(* IEC 61131-3 sources: AXOpen/src/components.keyence.vision/ctrl/src/Axo_IV3 (part 3) *)

            //*************************ToolResult_33*************************
            _retVal := Siemens.Simatic.DistributedIO.ReadData((Config.HWIDs.HwID_ToolResult_33) ,_data_in);
            IF _retVal > WORD#0 THEN
                Messenger.Activate(UINT#1638, eAxoMessageCategory#Error);
                Status.Error.Id := UINT#1638;
                RETURN;
            END_IF;

            _word.%B0 := _data_in[1];
            _word.%B1 := _data_in[0];
            Inputs.ToolResult_33.MatchingRate       :=  TO_UINT(_word);        // IW712
            _word.%B0 := _data_in[3];
            _word.%B1 := _data_in[2];
            Inputs.ToolResult_33.MatchingRateMAX    :=  TO_UINT(_word);        // IW714
            _word.%B0 := _data_in[5];
            _word.%B1 := _data_in[4];
            Inputs.ToolResult_33.MatchingRateMIN    :=  TO_UINT(_word);        // IW716
            _word.%B0 := _data_in[7];
            _word.%B1 := _data_in[6];
            Inputs.ToolResult_33.LowerThreshold     :=  TO_UINT(_word);        // IW718
            _word.%B0 := _data_in[9];
            _word.%B1 := _data_in[8];
            Inputs.ToolResult_33.UpperThreshold     :=  TO_UINT(_word);        // IW720
            _word.%B0 := _data_in[11];
            _word.%B1 := _data_in[10];
            Inputs.ToolResult_33.DecimalPointPosition:=  TO_UINT(_word);       // IW722
            _word.%B0 := _data_in[13];
            _word.%B1 := _data_in[12];
            Inputs.ToolResult_33.Data_1             :=  TO_UINT(_word);        // IW724
            _word.%B0 := _data_in[15];
            _word.%B1 := _data_in[14];
            Inputs.ToolResult_33.Data_2             :=  TO_UINT(_word);        // IW726
            _word.%B0 := _data_in[17];
            _word.%B1 := _data_in[16];
            Inputs.ToolResult_33.Data_3             :=  TO_UINT(_word);        // IW728
                                                                                    // IW730
            //***************************************************************

            //*************************ToolResult_34*************************
            _retVal := Siemens.Simatic.DistributedIO.ReadData((Config.HWIDs.HwID_ToolResult_34) ,_data_in);
            IF _retVal > WORD#0 THEN
                Messenger.Activate(UINT#1639, eAxoMessageCategory#Error);
                Status.Error.Id := UINT#1639;
                RETURN;
            END_IF;

            _word.%B0 := _data_in[1];
            _word.%B1 := _data_in[0];
            Inputs.ToolResult_34.MatchingRate       :=  TO_UINT(_word);        // IW732
            _word.%B0 := _data_in[3];
            _word.%B1 := _data_in[2];
            Inputs.ToolResult_34.MatchingRateMAX    :=  TO_UINT(_word);        // IW734
            _word.%B0 := _data_in[5];
            _word.%B1 := _data_in[4];
            Inputs.ToolResult_34.MatchingRateMIN    :=  TO_UINT(_word);        // IW736
            _word.%B0 := _data_in[7];
            _word.%B1 := _data_in[6];
            Inputs.ToolResult_34.LowerThreshold     :=  TO_UINT(_word);        // IW738
            _word.%B0 := _data_in[9];
            _word.%B1 := _data_in[8];
            Inputs.ToolResult_34.UpperThreshold     :=  TO_UINT(_word);        // IW740
            _word.%B0 := _data_in[11];
            _word.%B1 := _data_in[10];
            Inputs.ToolResult_34.DecimalPointPosition:=  TO_UINT(_word);       // IW742
            _word.%B0 := _data_in[13];
            _word.%B1 := _data_in[12];
            Inputs.ToolResult_34.Data_1             :=  TO_UINT(_word);        // IW744
            _word.%B0 := _data_in[15];
            _word.%B1 := _data_in[14];
            Inputs.ToolResult_34.Data_2             :=  TO_UINT(_word);        // IW746
            _word.%B0 := _data_in[17];
            _word.%B1 := _data_in[16];
            Inputs.ToolResult_34.Data_3             :=  TO_UINT(_word);        // IW748
                                                                                    // IW750
            //***************************************************************

            //*************************ToolResult_35*************************
            _retVal := Siemens.Simatic.DistributedIO.ReadData((Config.HWIDs.HwID_ToolResult_35) ,_data_in);
            IF _retVal > WORD#0 THEN
                Messenger.Activate(UINT#1640, eAxoMessageCategory#Error);
                Status.Error.Id := UINT#1640;
                RETURN;
            END_IF;

            _word.%B0 := _data_in[1];
            _word.%B1 := _data_in[0];
            Inputs.ToolResult_35.MatchingRate       :=  TO_UINT(_word);        // IW752
            _word.%B0 := _data_in[3];
            _word.%B1 := _data_in[2];
            Inputs.ToolResult_35.MatchingRateMAX    :=  TO_UINT(_word);        // IW754
            _word.%B0 := _data_in[5];
            _word.%B1 := _data_in[4];
            Inputs.ToolResult_35.MatchingRateMIN    :=  TO_UINT(_word);        // IW756
            _word.%B0 := _data_in[7];
            _word.%B1 := _data_in[6];
            Inputs.ToolResult_35.LowerThreshold     :=  TO_UINT(_word);        // IW758
            _word.%B0 := _data_in[9];
            _word.%B1 := _data_in[8];
            Inputs.ToolResult_35.UpperThreshold     :=  TO_UINT(_word);        // IW760
            _word.%B0 := _data_in[11];
            _word.%B1 := _data_in[10];
            Inputs.ToolResult_35.DecimalPointPosition:=  TO_UINT(_word);       // IW762
            _word.%B0 := _data_in[13];
            _word.%B1 := _data_in[12];
            Inputs.ToolResult_35.Data_1             :=  TO_UINT(_word);        // IW764
            _word.%B0 := _data_in[15];
            _word.%B1 := _data_in[14];
            Inputs.ToolResult_35.Data_2             :=  TO_UINT(_word);        // IW766
            _word.%B0 := _data_in[17];
            _word.%B1 := _data_in[16];
            Inputs.ToolResult_35.Data_3             :=  TO_UINT(_word);        // IW768
                                                                                    // IW770
            //***************************************************************

            //*************************ToolResult_36*************************
            _retVal := Siemens.Simatic.DistributedIO.ReadData((Config.HWIDs.HwID_ToolResult_36) ,_data_in);
            IF _retVal > WORD#0 THEN
                Messenger.Activate(UINT#1641, eAxoMessageCategory#Error);
                Status.Error.Id := UINT#1641;
                RETURN;
            END_IF;

            _word.%B0 := _data_in[1];
            _word.%B1 := _data_in[0];
            Inputs.ToolResult_36.MatchingRate       :=  TO_UINT(_word);        // IW772
            _word.%B0 := _data_in[3];
            _word.%B1 := _data_in[2];
            Inputs.ToolResult_36.MatchingRateMAX    :=  TO_UINT(_word);        // IW774
            _word.%B0 := _data_in[5];
            _word.%B1 := _data_in[4];
            Inputs.ToolResult_36.MatchingRateMIN    :=  TO_UINT(_word);        // IW776
            _word.%B0 := _data_in[7];
            _word.%B1 := _data_in[6];
            Inputs.ToolResult_36.LowerThreshold     :=  TO_UINT(_word);        // IW778
            _word.%B0 := _data_in[9];
            _word.%B1 := _data_in[8];
            Inputs.ToolResult_36.UpperThreshold     :=  TO_UINT(_word);        // IW780
            _word.%B0 := _data_in[11];
            _word.%B1 := _data_in[10];
            Inputs.ToolResult_36.DecimalPointPosition:=  TO_UINT(_word);       // IW782
            _word.%B0 := _data_in[13];
            _word.%B1 := _data_in[12];
            Inputs.ToolResult_36.Data_1             :=  TO_UINT(_word);        // IW784
            _word.%B0 := _data_in[15];
            _word.%B1 := _data_in[14];
            Inputs.ToolResult_36.Data_2             :=  TO_UINT(_word);        // IW786
            _word.%B0 := _data_in[17];
            _word.%B1 := _data_in[16];
            Inputs.ToolResult_36.Data_3             :=  TO_UINT(_word);        // IW788
                                                                                    // IW790
            //***************************************************************

            //*************************ToolResult_37*************************
            _retVal := Siemens.Simatic.DistributedIO.ReadData((Config.HWIDs.HwID_ToolResult_37) ,_data_in);
            IF _retVal > WORD#0 THEN
                Messenger.Activate(UINT#1642, eAxoMessageCategory#Error);
                Status.Error.Id := UINT#1642;
                RETURN;
            END_IF;

            _word.%B0 := _data_in[1];
            _word.%B1 := _data_in[0];
            Inputs.ToolResult_37.MatchingRate       :=  TO_UINT(_word);        // IW792
            _word.%B0 := _data_in[3];
            _word.%B1 := _data_in[2];
            Inputs.ToolResult_37.MatchingRateMAX    :=  TO_UINT(_word);        // IW794
            _word.%B0 := _data_in[5];
            _word.%B1 := _data_in[4];
            Inputs.ToolResult_37.MatchingRateMIN    :=  TO_UINT(_word);        // IW796
            _word.%B0 := _data_in[7];
            _word.%B1 := _data_in[6];
            Inputs.ToolResult_37.LowerThreshold     :=  TO_UINT(_word);        // IW798
            _word.%B0 := _data_in[9];
            _word.%B1 := _data_in[8];
            Inputs.ToolResult_37.UpperThreshold     :=  TO_UINT(_word);        // IW800
            _word.%B0 := _data_in[11];
            _word.%B1 := _data_in[10];
            Inputs.ToolResult_37.DecimalPointPosition:=  TO_UINT(_word);       // IW802
            _word.%B0 := _data_in[13];
            _word.%B1 := _data_in[12];
            Inputs.ToolResult_37.Data_1             :=  TO_UINT(_word);        // IW804
            _word.%B0 := _data_in[15];
            _word.%B1 := _data_in[14];
            Inputs.ToolResult_37.Data_2             :=  TO_UINT(_word);        // IW806
            _word.%B0 := _data_in[17];
            _word.%B1 := _data_in[16];
            Inputs.ToolResult_37.Data_3             :=  TO_UINT(_word);        // IW808
                                                                                    // IW810
            //***************************************************************

            //*************************ToolResult_38*************************
            _retVal := Siemens.Simatic.DistributedIO.ReadData((Config.HWIDs.HwID_ToolResult_38) ,_data_in);
            IF _retVal > WORD#0 THEN
                Messenger.Activate(UINT#1643, eAxoMessageCategory#Error);
                Status.Error.Id := UINT#1643;
                RETURN;
            END_IF;

            _word.%B0 := _data_in[1];
            _word.%B1 := _data_in[0];
            Inputs.ToolResult_38.MatchingRate       :=  TO_UINT(_word);        // IW812
            _word.%B0 := _data_in[3];
            _word.%B1 := _data_in[2];
            Inputs.ToolResult_38.MatchingRateMAX    :=  TO_UINT(_word);        // IW814
            _word.%B0 := _data_in[5];
            _word.%B1 := _data_in[4];
            Inputs.ToolResult_38.MatchingRateMIN    :=  TO_UINT(_word);        // IW816
            _word.%B0 := _data_in[7];
            _word.%B1 := _data_in[6];
            Inputs.ToolResult_38.LowerThreshold     :=  TO_UINT(_word);        // IW818
            _word.%B0 := _data_in[9];
            _word.%B1 := _data_in[8];
            Inputs.ToolResult_38.UpperThreshold     :=  TO_UINT(_word);        // IW820
            _word.%B0 := _data_in[11];
            _word.%B1 := _data_in[10];
            Inputs.ToolResult_38.DecimalPointPosition:=  TO_UINT(_word);       // IW822
            _word.%B0 := _data_in[13];
            _word.%B1 := _data_in[12];
            Inputs.ToolResult_38.Data_1             :=  TO_UINT(_word);        // IW824
            _word.%B0 := _data_in[15];
            _word.%B1 := _data_in[14];
            Inputs.ToolResult_38.Data_2             :=  TO_UINT(_word);        // IW826
            _word.%B0 := _data_in[17];
            _word.%B1 := _data_in[16];
            Inputs.ToolResult_38.Data_3             :=  TO_UINT(_word);        // IW828
                                                                                    // IW830
            //***************************************************************

            //*************************ToolResult_39*************************
            _retVal := Siemens.Simatic.DistributedIO.ReadData((Config.HWIDs.HwID_ToolResult_39) ,_data_in);
            IF _retVal > WORD#0 THEN
                Messenger.Activate(UINT#1644, eAxoMessageCategory#Error);
                Status.Error.Id := UINT#1644;
                RETURN;
            END_IF;

            _word.%B0 := _data_in[1];
            _word.%B1 := _data_in[0];
            Inputs.ToolResult_39.MatchingRate       :=  TO_UINT(_word);        // IW832
            _word.%B0 := _data_in[3];
            _word.%B1 := _data_in[2];
            Inputs.ToolResult_39.MatchingRateMAX    :=  TO_UINT(_word);        // IW834
            _word.%B0 := _data_in[5];
            _word.%B1 := _data_in[4];
            Inputs.ToolResult_39.MatchingRateMIN    :=  TO_UINT(_word);        // IW836
            _word.%B0 := _data_in[7];
            _word.%B1 := _data_in[6];
            Inputs.ToolResult_39.LowerThreshold     :=  TO_UINT(_word);        // IW838
            _word.%B0 := _data_in[9];
            _word.%B1 := _data_in[8];
            Inputs.ToolResult_39.UpperThreshold     :=  TO_UINT(_word);        // IW840
            _word.%B0 := _data_in[11];
            _word.%B1 := _data_in[10];
            Inputs.ToolResult_39.DecimalPointPosition:=  TO_UINT(_word);       // IW842
            _word.%B0 := _data_in[13];
            _word.%B1 := _data_in[12];
            Inputs.ToolResult_39.Data_1             :=  TO_UINT(_word);        // IW844
            _word.%B0 := _data_in[15];
            _word.%B1 := _data_in[14];
            Inputs.ToolResult_39.Data_2             :=  TO_UINT(_word);        // IW846
            _word.%B0 := _data_in[17];
            _word.%B1 := _data_in[16];
            Inputs.ToolResult_39.Data_3             :=  TO_UINT(_word);        // IW848
                                                                                    // IW850
            //***************************************************************

            //*************************ToolResult_40*************************
            _retVal := Siemens.Simatic.DistributedIO.ReadData((Config.HWIDs.HwID_ToolResult_40) ,_data_in);
            IF _retVal > WORD#0 THEN
                Messenger.Activate(UINT#1645, eAxoMessageCategory#Error);
                Status.Error.Id := UINT#1645;
                RETURN;
            END_IF;

            _word.%B0 := _data_in[1];
            _word.%B1 := _data_in[0];
            Inputs.ToolResult_40.MatchingRate       :=  TO_UINT(_word);        // IW852
            _word.%B0 := _data_in[3];
            _word.%B1 := _data_in[2];
            Inputs.ToolResult_40.MatchingRateMAX    :=  TO_UINT(_word);        // IW854
            _word.%B0 := _data_in[5];
            _word.%B1 := _data_in[4];
            Inputs.ToolResult_40.MatchingRateMIN    :=  TO_UINT(_word);        // IW856
            _word.%B0 := _data_in[7];
            _word.%B1 := _data_in[6];
            Inputs.ToolResult_40.LowerThreshold     :=  TO_UINT(_word);        // IW858
            _word.%B0 := _data_in[9];
            _word.%B1 := _data_in[8];
            Inputs.ToolResult_40.UpperThreshold     :=  TO_UINT(_word);        // IW860
            _word.%B0 := _data_in[11];
            _word.%B1 := _data_in[10];
            Inputs.ToolResult_40.DecimalPointPosition:=  TO_UINT(_word);       // IW862
            _word.%B0 := _data_in[13];
            _word.%B1 := _data_in[12];
            Inputs.ToolResult_40.Data_1             :=  TO_UINT(_word);        // IW864
            _word.%B0 := _data_in[15];
            _word.%B1 := _data_in[14];
            Inputs.ToolResult_40.Data_2             :=  TO_UINT(_word);        // IW866
            _word.%B0 := _data_in[17];
            _word.%B1 := _data_in[16];
            Inputs.ToolResult_40.Data_3             :=  TO_UINT(_word);        // IW868
                                                                                    // IW870
            //***************************************************************

            //*************************ToolResult_41*************************
            _retVal := Siemens.Simatic.DistributedIO.ReadData((Config.HWIDs.HwID_ToolResult_41) ,_data_in);
            IF _retVal > WORD#0 THEN
                Messenger.Activate(UINT#1646, eAxoMessageCategory#Error);
                Status.Error.Id := UINT#1646;
                RETURN;
            END_IF;

            _word.%B0 := _data_in[1];
            _word.%B1 := _data_in[0];
            Inputs.ToolResult_41.MatchingRate       :=  TO_UINT(_word);        // IW872
            _word.%B0 := _data_in[3];
            _word.%B1 := _data_in[2];
            Inputs.ToolResult_41.MatchingRateMAX    :=  TO_UINT(_word);        // IW874
            _word.%B0 := _data_in[5];
            _word.%B1 := _data_in[4];
            Inputs.ToolResult_41.MatchingRateMIN    :=  TO_UINT(_word);        // IW876
            _word.%B0 := _data_in[7];
            _word.%B1 := _data_in[6];
            Inputs.ToolResult_41.LowerThreshold     :=  TO_UINT(_word);        // IW878
            _word.%B0 := _data_in[9];
            _word.%B1 := _data_in[8];
            Inputs.ToolResult_41.UpperThreshold     :=  TO_UINT(_word);        // IW880
            _word.%B0 := _data_in[11];
            _word.%B1 := _data_in[10];
            Inputs.ToolResult_41.DecimalPointPosition:=  TO_UINT(_word);       // IW882
            _word.%B0 := _data_in[13];
            _word.%B1 := _data_in[12];
            Inputs.ToolResult_41.Data_1             :=  TO_UINT(_word);        // IW884
            _word.%B0 := _data_in[15];
            _word.%B1 := _data_in[14];
            Inputs.ToolResult_41.Data_2             :=  TO_UINT(_word);        // IW886
            _word.%B0 := _data_in[17];
            _word.%B1 := _data_in[16];
            Inputs.ToolResult_41.Data_3             :=  TO_UINT(_word);        // IW888
                                                                                    // IW890
            //***************************************************************

            //*************************ToolResult_42*************************
            _retVal := Siemens.Simatic.DistributedIO.ReadData((Config.HWIDs.HwID_ToolResult_42) ,_data_in);
            IF _retVal > WORD#0 THEN
                Messenger.Activate(UINT#1647, eAxoMessageCategory#Error);
                Status.Error.Id := UINT#1647;
                RETURN;
            END_IF;

            _word.%B0 := _data_in[1];
            _word.%B1 := _data_in[0];
            Inputs.ToolResult_42.MatchingRate       :=  TO_UINT(_word);        // IW892
            _word.%B0 := _data_in[3];
            _word.%B1 := _data_in[2];
            Inputs.ToolResult_42.MatchingRateMAX    :=  TO_UINT(_word);        // IW894
            _word.%B0 := _data_in[5];
            _word.%B1 := _data_in[4];
            Inputs.ToolResult_42.MatchingRateMIN    :=  TO_UINT(_word);        // IW896
            _word.%B0 := _data_in[7];
            _word.%B1 := _data_in[6];
            Inputs.ToolResult_42.LowerThreshold     :=  TO_UINT(_word);        // IW898
            _word.%B0 := _data_in[9];
            _word.%B1 := _data_in[8];
            Inputs.ToolResult_42.UpperThreshold     :=  TO_UINT(_word);        // IW900
            _word.%B0 := _data_in[11];
            _word.%B1 := _data_in[10];
            Inputs.ToolResult_42.DecimalPointPosition:=  TO_UINT(_word);       // IW902
            _word.%B0 := _data_in[13];
            _word.%B1 := _data_in[12];
            Inputs.ToolResult_42.Data_1             :=  TO_UINT(_word);        // IW904
            _word.%B0 := _data_in[15];
            _word.%B1 := _data_in[14];
            Inputs.ToolResult_42.Data_2             :=  TO_UINT(_word);        // IW906
            _word.%B0 := _data_in[17];
            _word.%B1 := _data_in[16];
            Inputs.ToolResult_42.Data_3             :=  TO_UINT(_word);        // IW908
                                                                                    // IW910
            //***************************************************************

            //*************************ToolResult_43*************************
            _retVal := Siemens.Simatic.DistributedIO.ReadData((Config.HWIDs.HwID_ToolResult_43) ,_data_in);
            IF _retVal > WORD#0 THEN
                Messenger.Activate(UINT#1648, eAxoMessageCategory#Error);
                Status.Error.Id := UINT#1648;
                RETURN;
            END_IF;

            _word.%B0 := _data_in[1];
            _word.%B1 := _data_in[0];
            Inputs.ToolResult_43.MatchingRate       :=  TO_UINT(_word);        // IW912
            _word.%B0 := _data_in[3];
            _word.%B1 := _data_in[2];
            Inputs.ToolResult_43.MatchingRateMAX    :=  TO_UINT(_word);        // IW914
            _word.%B0 := _data_in[5];
            _word.%B1 := _data_in[4];
            Inputs.ToolResult_43.MatchingRateMIN    :=  TO_UINT(_word);        // IW916
            _word.%B0 := _data_in[7];
            _word.%B1 := _data_in[6];
            Inputs.ToolResult_43.LowerThreshold     :=  TO_UINT(_word);        // IW918
            _word.%B0 := _data_in[9];
            _word.%B1 := _data_in[8];
            Inputs.ToolResult_43.UpperThreshold     :=  TO_UINT(_word);        // IW920
            _word.%B0 := _data_in[11];
            _word.%B1 := _data_in[10];
            Inputs.ToolResult_43.DecimalPointPosition:=  TO_UINT(_word);       // IW922
            _word.%B0 := _data_in[13];
            _word.%B1 := _data_in[12];
            Inputs.ToolResult_43.Data_1             :=  TO_UINT(_word);        // IW924
            _word.%B0 := _data_in[15];
            _word.%B1 := _data_in[14];
            Inputs.ToolResult_43.Data_2             :=  TO_UINT(_word);        // IW926
            _word.%B0 := _data_in[17];
            _word.%B1 := _data_in[16];
            Inputs.ToolResult_43.Data_3             :=  TO_UINT(_word);        // IW928
                                                                                    // IW930
            //***************************************************************

            //*************************ToolResult_44*************************
            _retVal := Siemens.Simatic.DistributedIO.ReadData((Config.HWIDs.HwID_ToolResult_44) ,_data_in);
            IF _retVal > WORD#0 THEN
                Messenger.Activate(UINT#1649, eAxoMessageCategory#Error);
                Status.Error.Id := UINT#1649;
                RETURN;
            END_IF;

            _word.%B0 := _data_in[1];
            _word.%B1 := _data_in[0];
            Inputs.ToolResult_44.MatchingRate       :=  TO_UINT(_word);        // IW932
            _word.%B0 := _data_in[3];
            _word.%B1 := _data_in[2];
            Inputs.ToolResult_44.MatchingRateMAX    :=  TO_UINT(_word);        // IW934
            _word.%B0 := _data_in[5];
            _word.%B1 := _data_in[4];
            Inputs.ToolResult_44.MatchingRateMIN    :=  TO_UINT(_word);        // IW936
            _word.%B0 := _data_in[7];
            _word.%B1 := _data_in[6];
            Inputs.ToolResult_44.LowerThreshold     :=  TO_UINT(_word);        // IW938
            _word.%B0 := _data_in[9];
            _word.%B1 := _data_in[8];
            Inputs.ToolResult_44.UpperThreshold     :=  TO_UINT(_word);        // IW940
            _word.%B0 := _data_in[11];
            _word.%B1 := _data_in[10];
            Inputs.ToolResult_44.DecimalPointPosition:=  TO_UINT(_word);       // IW942
            _word.%B0 := _data_in[13];
            _word.%B1 := _data_in[12];
            Inputs.ToolResult_44.Data_1             :=  TO_UINT(_word);        // IW944
            _word.%B0 := _data_in[15];
            _word.%B1 := _data_in[14];
            Inputs.ToolResult_44.Data_2             :=  TO_UINT(_word);        // IW946
            _word.%B0 := _data_in[17];
            _word.%B1 := _data_in[16];
            Inputs.ToolResult_44.Data_3             :=  TO_UINT(_word);        // IW948
                                                                                    // IW950
            //***************************************************************

            //*************************ToolResult_45*************************
            _retVal := Siemens.Simatic.DistributedIO.ReadData((Config.HWIDs.HwID_ToolResult_45) ,_data_in);
            IF _retVal > WORD#0 THEN
                Messenger.Activate(UINT#1650, eAxoMessageCategory#Error);
                Status.Error.Id := UINT#1650;
                RETURN;
            END_IF;

            _word.%B0 := _data_in[1];
            _word.%B1 := _data_in[0];
            Inputs.ToolResult_45.MatchingRate       :=  TO_UINT(_word);        // IW952
            _word.%B0 := _data_in[3];
            _word.%B1 := _data_in[2];
            Inputs.ToolResult_45.MatchingRateMAX    :=  TO_UINT(_word);        // IW954
            _word.%B0 := _data_in[5];
            _word.%B1 := _data_in[4];
            Inputs.ToolResult_45.MatchingRateMIN    :=  TO_UINT(_word);        // IW956
            _word.%B0 := _data_in[7];
            _word.%B1 := _data_in[6];
            Inputs.ToolResult_45.LowerThreshold     :=  TO_UINT(_word);        // IW958
            _word.%B0 := _data_in[9];
            _word.%B1 := _data_in[8];
            Inputs.ToolResult_45.UpperThreshold     :=  TO_UINT(_word);        // IW960
            _word.%B0 := _data_in[11];
            _word.%B1 := _data_in[10];
            Inputs.ToolResult_45.DecimalPointPosition:=  TO_UINT(_word);       // IW962
            _word.%B0 := _data_in[13];
            _word.%B1 := _data_in[12];
            Inputs.ToolResult_45.Data_1             :=  TO_UINT(_word);        // IW964
            _word.%B0 := _data_in[15];
            _word.%B1 := _data_in[14];
            Inputs.ToolResult_45.Data_2             :=  TO_UINT(_word);        // IW966
            _word.%B0 := _data_in[17];
            _word.%B1 := _data_in[16];
            Inputs.ToolResult_45.Data_3             :=  TO_UINT(_word);        // IW968
                                                                                    // IW970
            //***************************************************************

            //*************************ToolResult_46*************************
            _retVal := Siemens.Simatic.DistributedIO.ReadData((Config.HWIDs.HwID_ToolResult_46) ,_data_in);
            IF _retVal > WORD#0 THEN
                Messenger.Activate(UINT#1651, eAxoMessageCategory#Error);
                Status.Error.Id := UINT#1651;
                RETURN;
            END_IF;

            _word.%B0 := _data_in[1];
            _word.%B1 := _data_in[0];
            Inputs.ToolResult_46.MatchingRate       :=  TO_UINT(_word);        // IW972
            _word.%B0 := _data_in[3];
            _word.%B1 := _data_in[2];
            Inputs.ToolResult_46.MatchingRateMAX    :=  TO_UINT(_word);        // IW974
            _word.%B0 := _data_in[5];
            _word.%B1 := _data_in[4];
            Inputs.ToolResult_46.MatchingRateMIN    :=  TO_UINT(_word);        // IW976
            _word.%B0 := _data_in[7];
            _word.%B1 := _data_in[6];
            Inputs.ToolResult_46.LowerThreshold     :=  TO_UINT(_word);        // IW978
            _word.%B0 := _data_in[9];
            _word.%B1 := _data_in[8];
            Inputs.ToolResult_46.UpperThreshold     :=  TO_UINT(_word);        // IW980
            _word.%B0 := _data_in[11];
            _word.%B1 := _data_in[10];
            Inputs.ToolResult_46.DecimalPointPosition:=  TO_UINT(_word);       // IW982
            _word.%B0 := _data_in[13];
            _word.%B1 := _data_in[12];
            Inputs.ToolResult_46.Data_1             :=  TO_UINT(_word);        // IW984
            _word.%B0 := _data_in[15];
            _word.%B1 := _data_in[14];
            Inputs.ToolResult_46.Data_2             :=  TO_UINT(_word);        // IW986
            _word.%B0 := _data_in[17];
            _word.%B1 := _data_in[16];
            Inputs.ToolResult_46.Data_3             :=  TO_UINT(_word);        // IW988
                                                                                    // IW990
            //***************************************************************

            //*************************ToolResult_47*************************
            _retVal := Siemens.Simatic.DistributedIO.ReadData((Config.HWIDs.HwID_ToolResult_47) ,_data_in);
            IF _retVal > WORD#0 THEN
                Messenger.Activate(UINT#1652, eAxoMessageCategory#Error);
                Status.Error.Id := UINT#1652;
                RETURN;
            END_IF;

            _word.%B0 := _data_in[1];
            _word.%B1 := _data_in[0];
            Inputs.ToolResult_47.MatchingRate       :=  TO_UINT(_word);        // IW992
            _word.%B0 := _data_in[3];
            _word.%B1 := _data_in[2];
            Inputs.ToolResult_47.MatchingRateMAX    :=  TO_UINT(_word);        // IW994
            _word.%B0 := _data_in[5];
            _word.%B1 := _data_in[4];
            Inputs.ToolResult_47.MatchingRateMIN    :=  TO_UINT(_word);        // IW996
            _word.%B0 := _data_in[7];
            _word.%B1 := _data_in[6];
            Inputs.ToolResult_47.LowerThreshold     :=  TO_UINT(_word);        // IW998
            _word.%B0 := _data_in[9];
            _word.%B1 := _data_in[8];
            Inputs.ToolResult_47.UpperThreshold     :=  TO_UINT(_word);        // IW1000
            _word.%B0 := _data_in[11];
            _word.%B1 := _data_in[10];
            Inputs.ToolResult_47.DecimalPointPosition:=  TO_UINT(_word);       // IW1002
            _word.%B0 := _data_in[13];
            _word.%B1 := _data_in[12];
            Inputs.ToolResult_47.Data_1             :=  TO_UINT(_word);        // IW1004
            _word.%B0 := _data_in[15];
            _word.%B1 := _data_in[14];
            Inputs.ToolResult_47.Data_2             :=  TO_UINT(_word);        // IW1006
            _word.%B0 := _data_in[17];
            _word.%B1 := _data_in[16];
            Inputs.ToolResult_47.Data_3             :=  TO_UINT(_word);        // IW1008
                                                                                    // IW1010
            //***************************************************************

            //*************************ToolResult_48*************************
            _retVal := Siemens.Simatic.DistributedIO.ReadData((Config.HWIDs.HwID_ToolResult_48) ,_data_in);
            IF _retVal > WORD#0 THEN
                Messenger.Activate(UINT#1653, eAxoMessageCategory#Error);
                Status.Error.Id := UINT#1653;
                RETURN;
            END_IF;

            _word.%B0 := _data_in[1];
            _word.%B1 := _data_in[0];
            Inputs.ToolResult_48.MatchingRate       :=  TO_UINT(_word);        // IW1012
            _word.%B0 := _data_in[3];
            _word.%B1 := _data_in[2];
            Inputs.ToolResult_48.MatchingRateMAX    :=  TO_UINT(_word);        // IW1014
            _word.%B0 := _data_in[5];
            _word.%B1 := _data_in[4];
            Inputs.ToolResult_48.MatchingRateMIN    :=  TO_UINT(_word);        // IW1016
            _word.%B0 := _data_in[7];
            _word.%B1 := _data_in[6];
            Inputs.ToolResult_48.LowerThreshold     :=  TO_UINT(_word);        // IW1018
            _word.%B0 := _data_in[9];
            _word.%B1 := _data_in[8];
            Inputs.ToolResult_48.UpperThreshold     :=  TO_UINT(_word);        // IW1020
            _word.%B0 := _data_in[11];
            _word.%B1 := _data_in[10];
            Inputs.ToolResult_48.DecimalPointPosition:=  TO_UINT(_word);       // IW1022
            _word.%B0 := _data_in[13];
            _word.%B1 := _data_in[12];
            Inputs.ToolResult_48.Data_1             :=  TO_UINT(_word);        // IW1024
            _word.%B0 := _data_in[15];
            _word.%B1 := _data_in[14];
            Inputs.ToolResult_48.Data_2             :=  TO_UINT(_word);        // IW1026
            _word.%B0 := _data_in[17];
            _word.%B1 := _data_in[16];
            Inputs.ToolResult_48.Data_3             :=  TO_UINT(_word);        // IW1028
                                                                                    // IW1030
            //***************************************************************

            //*************************ToolResult_49*************************
            _retVal := Siemens.Simatic.DistributedIO.ReadData((Config.HWIDs.HwID_ToolResult_49) ,_data_in);
            IF _retVal > WORD#0 THEN
                Messenger.Activate(UINT#1654, eAxoMessageCategory#Error);
                Status.Error.Id := UINT#1654;
                RETURN;
            END_IF;

            _word.%B0 := _data_in[1];
            _word.%B1 := _data_in[0];
            Inputs.ToolResult_49.MatchingRate       :=  TO_UINT(_word);        // IW1032
            _word.%B0 := _data_in[3];
            _word.%B1 := _data_in[2];
            Inputs.ToolResult_49.MatchingRateMAX    :=  TO_UINT(_word);        // IW1034
            _word.%B0 := _data_in[5];
            _word.%B1 := _data_in[4];
            Inputs.ToolResult_49.MatchingRateMIN    :=  TO_UINT(_word);        // IW1036
            _word.%B0 := _data_in[7];
            _word.%B1 := _data_in[6];
            Inputs.ToolResult_49.LowerThreshold     :=  TO_UINT(_word);        // IW1038
            _word.%B0 := _data_in[9];
            _word.%B1 := _data_in[8];
            Inputs.ToolResult_49.UpperThreshold     :=  TO_UINT(_word);        // IW1040
            _word.%B0 := _data_in[11];
            _word.%B1 := _data_in[10];
            Inputs.ToolResult_49.DecimalPointPosition:=  TO_UINT(_word);       // IW1042
            _word.%B0 := _data_in[13];
            _word.%B1 := _data_in[12];
            Inputs.ToolResult_49.Data_1             :=  TO_UINT(_word);        // IW1044
            _word.%B0 := _data_in[15];
            _word.%B1 := _data_in[14];
            Inputs.ToolResult_49.Data_2             :=  TO_UINT(_word);        // IW1046
            _word.%B0 := _data_in[17];
            _word.%B1 := _data_in[16];
            Inputs.ToolResult_49.Data_3             :=  TO_UINT(_word);        // IW1048
                                                                                    // IW1050
            //***************************************************************

            //*************************ToolResult_50*************************
            _retVal := Siemens.Simatic.DistributedIO.ReadData((Config.HWIDs.HwID_ToolResult_50) ,_data_in);
            IF _retVal > WORD#0 THEN
                Messenger.Activate(UINT#1655, eAxoMessageCategory#Error);
                Status.Error.Id := UINT#1655;
                RETURN;
            END_IF;

            _word.%B0 := _data_in[1];
            _word.%B1 := _data_in[0];
            Inputs.ToolResult_50.MatchingRate       :=  TO_UINT(_word);        // IW1052
            _word.%B0 := _data_in[3];
            _word.%B1 := _data_in[2];
            Inputs.ToolResult_50.MatchingRateMAX    :=  TO_UINT(_word);        // IW1054
            _word.%B0 := _data_in[5];
            _word.%B1 := _data_in[4];
            Inputs.ToolResult_50.MatchingRateMIN    :=  TO_UINT(_word);        // IW1056
            _word.%B0 := _data_in[7];
            _word.%B1 := _data_in[6];
            Inputs.ToolResult_50.LowerThreshold     :=  TO_UINT(_word);        // IW1058
            _word.%B0 := _data_in[9];
            _word.%B1 := _data_in[8];
            Inputs.ToolResult_50.UpperThreshold     :=  TO_UINT(_word);        // IW1060
            _word.%B0 := _data_in[11];
            _word.%B1 := _data_in[10];
            Inputs.ToolResult_50.DecimalPointPosition:=  TO_UINT(_word);       // IW1062
            _word.%B0 := _data_in[13];
            _word.%B1 := _data_in[12];
            Inputs.ToolResult_50.Data_1             :=  TO_UINT(_word);        // IW1064
            _word.%B0 := _data_in[15];
            _word.%B1 := _data_in[14];
            Inputs.ToolResult_50.Data_2             :=  TO_UINT(_word);        // IW1066
            _word.%B0 := _data_in[17];
            _word.%B1 := _data_in[16];
            Inputs.ToolResult_50.Data_3             :=  TO_UINT(_word);        // IW1068
                                                                                    // IW1070
            //***************************************************************

            //*************************ToolResult_51*************************
            _retVal := Siemens.Simatic.DistributedIO.ReadData((Config.HWIDs.HwID_ToolResult_51) ,_data_in);
            IF _retVal > WORD#0 THEN
                Messenger.Activate(UINT#1656, eAxoMessageCategory#Error);
                Status.Error.Id := UINT#1656;
                RETURN;
            END_IF;

            _word.%B0 := _data_in[1];
            _word.%B1 := _data_in[0];
            Inputs.ToolResult_51.MatchingRate       :=  TO_UINT(_word);        // IW1072
            _word.%B0 := _data_in[3];
            _word.%B1 := _data_in[2];
            Inputs.ToolResult_51.MatchingRateMAX    :=  TO_UINT(_word);        // IW1074
            _word.%B0 := _data_in[5];
            _word.%B1 := _data_in[4];
            Inputs.ToolResult_51.MatchingRateMIN    :=  TO_UINT(_word);        // IW1076
            _word.%B0 := _data_in[7];
            _word.%B1 := _data_in[6];
            Inputs.ToolResult_51.LowerThreshold     :=  TO_UINT(_word);        // IW1078
            _word.%B0 := _data_in[9];
            _word.%B1 := _data_in[8];
            Inputs.ToolResult_51.UpperThreshold     :=  TO_UINT(_word);        // IW1080
            _word.%B0 := _data_in[11];
            _word.%B1 := _data_in[10];
            Inputs.ToolResult_51.DecimalPointPosition:=  TO_UINT(_word);       // IW1082
            _word.%B0 := _data_in[13];
            _word.%B1 := _data_in[12];
            Inputs.ToolResult_51.Data_1             :=  TO_UINT(_word);        // IW1084
            _word.%B0 := _data_in[15];
            _word.%B1 := _data_in[14];
            Inputs.ToolResult_51.Data_2             :=  TO_UINT(_word);        // IW1086
            _word.%B0 := _data_in[17];
            _word.%B1 := _data_in[16];
            Inputs.ToolResult_51.Data_3             :=  TO_UINT(_word);        // IW1088
                                                                                    // IW1090
            //***************************************************************

            //*************************ToolResult_52*************************
            _retVal := Siemens.Simatic.DistributedIO.ReadData((Config.HWIDs.HwID_ToolResult_52) ,_data_in);
            IF _retVal > WORD#0 THEN
                Messenger.Activate(UINT#1657, eAxoMessageCategory#Error);
                Status.Error.Id := UINT#1657;
                RETURN;
            END_IF;

            _word.%B0 := _data_in[1];
            _word.%B1 := _data_in[0];
            Inputs.ToolResult_52.MatchingRate       :=  TO_UINT(_word);        // IW1092
            _word.%B0 := _data_in[3];
            _word.%B1 := _data_in[2];
            Inputs.ToolResult_52.MatchingRateMAX    :=  TO_UINT(_word);        // IW1094
            _word.%B0 := _data_in[5];
            _word.%B1 := _data_in[4];
            Inputs.ToolResult_52.MatchingRateMIN    :=  TO_UINT(_word);        // IW1096
            _word.%B0 := _data_in[7];
            _word.%B1 := _data_in[6];
            Inputs.ToolResult_52.LowerThreshold     :=  TO_UINT(_word);        // IW1098
            _word.%B0 := _data_in[9];
            _word.%B1 := _data_in[8];
            Inputs.ToolResult_52.UpperThreshold     :=  TO_UINT(_word);        // IW1100
            _word.%B0 := _data_in[11];
            _word.%B1 := _data_in[10];
            Inputs.ToolResult_52.DecimalPointPosition:=  TO_UINT(_word);       // IW1102
            _word.%B0 := _data_in[13];
            _word.%B1 := _data_in[12];
            Inputs.ToolResult_52.Data_1             :=  TO_UINT(_word);        // IW1104
            _word.%B0 := _data_in[15];
            _word.%B1 := _data_in[14];
            Inputs.ToolResult_52.Data_2             :=  TO_UINT(_word);        // IW1106
            _word.%B0 := _data_in[17];
            _word.%B1 := _data_in[16];
            Inputs.ToolResult_52.Data_3             :=  TO_UINT(_word);        // IW1108
                                                                                    // IW1110
            //***************************************************************

            //*************************ToolResult_53*************************
            _retVal := Siemens.Simatic.DistributedIO.ReadData((Config.HWIDs.HwID_ToolResult_53) ,_data_in);
            IF _retVal > WORD#0 THEN
                Messenger.Activate(UINT#1658, eAxoMessageCategory#Error);
                Status.Error.Id := UINT#1658;
                RETURN;
            END_IF;

            _word.%B0 := _data_in[1];
            _word.%B1 := _data_in[0];
            Inputs.ToolResult_53.MatchingRate       :=  TO_UINT(_word);        // IW1112
            _word.%B0 := _data_in[3];
            _word.%B1 := _data_in[2];
            Inputs.ToolResult_53.MatchingRateMAX    :=  TO_UINT(_word);        // IW1114
            _word.%B0 := _data_in[5];
            _word.%B1 := _data_in[4];
            Inputs.ToolResult_53.MatchingRateMIN    :=  TO_UINT(_word);        // IW1116
            _word.%B0 := _data_in[7];
            _word.%B1 := _data_in[6];
            Inputs.ToolResult_53.LowerThreshold     :=  TO_UINT(_word);        // IW1118
            _word.%B0 := _data_in[9];
            _word.%B1 := _data_in[8];
            Inputs.ToolResult_53.UpperThreshold     :=  TO_UINT(_word);        // IW1120
            _word.%B0 := _data_in[11];
            _word.%B1 := _data_in[10];
            Inputs.ToolResult_53.DecimalPointPosition:=  TO_UINT(_word);       // IW1122
            _word.%B0 := _data_in[13];
            _word.%B1 := _data_in[12];
            Inputs.ToolResult_53.Data_1             :=  TO_UINT(_word);        // IW1124
            _word.%B0 := _data_in[15];
            _word.%B1 := _data_in[14];
            Inputs.ToolResult_53.Data_2             :=  TO_UINT(_word);        // IW1126
            _word.%B0 := _data_in[17];
            _word.%B1 := _data_in[16];
            Inputs.ToolResult_53.Data_3             :=  TO_UINT(_word);        // IW1128
                                                                                    // IW1130
            //***************************************************************

            //*************************ToolResult_54*************************
            _retVal := Siemens.Simatic.DistributedIO.ReadData((Config.HWIDs.HwID_ToolResult_54) ,_data_in);
            IF _retVal > WORD#0 THEN
                Messenger.Activate(UINT#1659, eAxoMessageCategory#Error);
                Status.Error.Id := UINT#1659;
                RETURN;
            END_IF;

            _word.%B0 := _data_in[1];
            _word.%B1 := _data_in[0];
            Inputs.ToolResult_54.MatchingRate       :=  TO_UINT(_word);        // IW1132
            _word.%B0 := _data_in[3];
            _word.%B1 := _data_in[2];
            Inputs.ToolResult_54.MatchingRateMAX    :=  TO_UINT(_word);        // IW1134
            _word.%B0 := _data_in[5];
            _word.%B1 := _data_in[4];
            Inputs.ToolResult_54.MatchingRateMIN    :=  TO_UINT(_word);        // IW1136
            _word.%B0 := _data_in[7];
            _word.%B1 := _data_in[6];
            Inputs.ToolResult_54.LowerThreshold     :=  TO_UINT(_word);        // IW1138
            _word.%B0 := _data_in[9];
            _word.%B1 := _data_in[8];
            Inputs.ToolResult_54.UpperThreshold     :=  TO_UINT(_word);        // IW1140
            _word.%B0 := _data_in[11];
            _word.%B1 := _data_in[10];
            Inputs.ToolResult_54.DecimalPointPosition:=  TO_UINT(_word);       // IW1142
            _word.%B0 := _data_in[13];
            _word.%B1 := _data_in[12];
            Inputs.ToolResult_54.Data_1             :=  TO_UINT(_word);        // IW1144
            _word.%B0 := _data_in[15];
            _word.%B1 := _data_in[14];
            Inputs.ToolResult_54.Data_2             :=  TO_UINT(_word);        // IW1146
            _word.%B0 := _data_in[17];
            _word.%B1 := _data_in[16];
            Inputs.ToolResult_54.Data_3             :=  TO_UINT(_word);        // IW1148
                                                                                    // IW1150
            //***************************************************************

            //*************************ToolResult_55*************************
            _retVal := Siemens.Simatic.DistributedIO.ReadData((Config.HWIDs.HwID_ToolResult_55) ,_data_in);
            IF _retVal > WORD#0 THEN
                Messenger.Activate(UINT#1660, eAxoMessageCategory#Error);
                Status.Error.Id := UINT#1660;
                RETURN;
            END_IF;

            _word.%B0 := _data_in[1];
            _word.%B1 := _data_in[0];
            Inputs.ToolResult_55.MatchingRate       :=  TO_UINT(_word);        // IW1152
            _word.%B0 := _data_in[3];
            _word.%B1 := _data_in[2];
            Inputs.ToolResult_55.MatchingRateMAX    :=  TO_UINT(_word);        // IW1154
            _word.%B0 := _data_in[5];
            _word.%B1 := _data_in[4];
            Inputs.ToolResult_55.MatchingRateMIN    :=  TO_UINT(_word);        // IW1156
            _word.%B0 := _data_in[7];
            _word.%B1 := _data_in[6];
            Inputs.ToolResult_55.LowerThreshold     :=  TO_UINT(_word);        // IW1158
            _word.%B0 := _data_in[9];
            _word.%B1 := _data_in[8];
            Inputs.ToolResult_55.UpperThreshold     :=  TO_UINT(_word);        // IW1160
            _word.%B0 := _data_in[11];
            _word.%B1 := _data_in[10];
            Inputs.ToolResult_55.DecimalPointPosition:=  TO_UINT(_word);       // IW1162
            _word.%B0 := _data_in[13];
            _word.%B1 := _data_in[12];
            Inputs.ToolResult_55.Data_1             :=  TO_UINT(_word);        // IW1164
            _word.%B0 := _data_in[15];
            _word.%B1 := _data_in[14];
            Inputs.ToolResult_55.Data_2             :=  TO_UINT(_word);        // IW1166
            _word.%B0 := _data_in[17];
            _word.%B1 := _data_in[16];
            Inputs.ToolResult_55.Data_3             :=  TO_UINT(_word);        // IW1168
                                                                                    // IW1170
            //***************************************************************

            //*************************ToolResult_56*************************
            _retVal := Siemens.Simatic.DistributedIO.ReadData((Config.HWIDs.HwID_ToolResult_56) ,_data_in);
            IF _retVal > WORD#0 THEN
                Messenger.Activate(UINT#1661, eAxoMessageCategory#Error);
                Status.Error.Id := UINT#1661;
                RETURN;
            END_IF;

            _word.%B0 := _data_in[1];
            _word.%B1 := _data_in[0];
            Inputs.ToolResult_56.MatchingRate       :=  TO_UINT(_word);        // IW1172
            _word.%B0 := _data_in[3];
            _word.%B1 := _data_in[2];
            Inputs.ToolResult_56.MatchingRateMAX    :=  TO_UINT(_word);        // IW1174
            _word.%B0 := _data_in[5];
            _word.%B1 := _data_in[4];
            Inputs.ToolResult_56.MatchingRateMIN    :=  TO_UINT(_word);        // IW1176
            _word.%B0 := _data_in[7];
            _word.%B1 := _data_in[6];
            Inputs.ToolResult_56.LowerThreshold     :=  TO_UINT(_word);        // IW1178
            _word.%B0 := _data_in[9];
            _word.%B1 := _data_in[8];
            Inputs.ToolResult_56.UpperThreshold     :=  TO_UINT(_word);        // IW1180
            _word.%B0 := _data_in[11];
            _word.%B1 := _data_in[10];
            Inputs.ToolResult_56.DecimalPointPosition:=  TO_UINT(_word);       // IW1182
            _word.%B0 := _data_in[13];
            _word.%B1 := _data_in[12];
            Inputs.ToolResult_56.Data_1             :=  TO_UINT(_word);        // IW1184
            _word.%B0 := _data_in[15];
            _word.%B1 := _data_in[14];
            Inputs.ToolResult_56.Data_2             :=  TO_UINT(_word);        // IW1186
            _word.%B0 := _data_in[17];
            _word.%B1 := _data_in[16];
            Inputs.ToolResult_56.Data_3             :=  TO_UINT(_word);        // IW1188
                                                                                    // IW1190
            //***************************************************************

            //*************************ToolResult_57*************************
            _retVal := Siemens.Simatic.DistributedIO.ReadData((Config.HWIDs.HwID_ToolResult_57) ,_data_in);
            IF _retVal > WORD#0 THEN
                Messenger.Activate(UINT#1662, eAxoMessageCategory#Error);
                Status.Error.Id := UINT#1662;
                RETURN;
            END_IF;

            _word.%B0 := _data_in[1];
            _word.%B1 := _data_in[0];
            Inputs.ToolResult_57.MatchingRate       :=  TO_UINT(_word);        // IW1192
            _word.%B0 := _data_in[3];
            _word.%B1 := _data_in[2];
            Inputs.ToolResult_57.MatchingRateMAX    :=  TO_UINT(_word);        // IW1194
            _word.%B0 := _data_in[5];
            _word.%B1 := _data_in[4];
            Inputs.ToolResult_57.MatchingRateMIN    :=  TO_UINT(_word);        // IW1196
            _word.%B0 := _data_in[7];
            _word.%B1 := _data_in[6];
            Inputs.ToolResult_57.LowerThreshold     :=  TO_UINT(_word);        // IW1198
            _word.%B0 := _data_in[9];
            _word.%B1 := _data_in[8];
            Inputs.ToolResult_57.UpperThreshold     :=  TO_UINT(_word);        // IW1200
            _word.%B0 := _data_in[11];
            _word.%B1 := _data_in[10];
            Inputs.ToolResult_57.DecimalPointPosition:=  TO_UINT(_word);       // IW1202
            _word.%B0 := _data_in[13];
            _word.%B1 := _data_in[12];
            Inputs.ToolResult_57.Data_1             :=  TO_UINT(_word);        // IW1204
            _word.%B0 := _data_in[15];
            _word.%B1 := _data_in[14];
            Inputs.ToolResult_57.Data_2             :=  TO_UINT(_word);        // IW1206
            _word.%B0 := _data_in[17];
            _word.%B1 := _data_in[16];
            Inputs.ToolResult_57.Data_3             :=  TO_UINT(_word);        // IW1208
                                                                                    // IW1210
            //***************************************************************

            //*************************ToolResult_58*************************
            _retVal := Siemens.Simatic.DistributedIO.ReadData((Config.HWIDs.HwID_ToolResult_58) ,_data_in);
            IF _retVal > WORD#0 THEN
                Messenger.Activate(UINT#1663, eAxoMessageCategory#Error);
                Status.Error.Id := UINT#1663;
                RETURN;
            END_IF;

            _word.%B0 := _data_in[1];
            _word.%B1 := _data_in[0];
            Inputs.ToolResult_58.MatchingRate       :=  TO_UINT(_word);        // IW1212
            _word.%B0 := _data_in[3];
            _word.%B1 := _data_in[2];
            Inputs.ToolResult_58.MatchingRateMAX    :=  TO_UINT(_word);        // IW1214
            _word.%B0 := _data_in[5];
            _word.%B1 := _data_in[4];
            Inputs.ToolResult_58.MatchingRateMIN    :=  TO_UINT(_word);        // IW1216
            _word.%B0 := _data_in[7];
            _word.%B1 := _data_in[6];
            Inputs.ToolResult_58.LowerThreshold     :=  TO_UINT(_word);        // IW1218
            _word.%B0 := _data_in[9];
            _word.%B1 := _data_in[8];
            Inputs.ToolResult_58.UpperThreshold     :=  TO_UINT(_word);        // IW1220
            _word.%B0 := _data_in[11];
            _word.%B1 := _data_in[10];
            Inputs.ToolResult_58.DecimalPointPosition:=  TO_UINT(_word);       // IW1222
            _word.%B0 := _data_in[13];
            _word.%B1 := _data_in[12];
            Inputs.ToolResult_58.Data_1             :=  TO_UINT(_word);        // IW1224
            _word.%B0 := _data_in[15];
            _word.%B1 := _data_in[14];
            Inputs.ToolResult_58.Data_2             :=  TO_UINT(_word);        // IW1226
            _word.%B0 := _data_in[17];
            _word.%B1 := _data_in[16];
            Inputs.ToolResult_58.Data_3             :=  TO_UINT(_word);        // IW1228
                                                                                    // IW1230
            //***************************************************************

            //*************************ToolResult_59*************************
            _retVal := Siemens.Simatic.DistributedIO.ReadData((Config.HWIDs.HwID_ToolResult_59) ,_data_in);
            IF _retVal > WORD#0 THEN
                Messenger.Activate(UINT#1664, eAxoMessageCategory#Error);
                Status.Error.Id := UINT#1664;
                RETURN;
            END_IF;

            _word.%B0 := _data_in[1];
            _word.%B1 := _data_in[0];
            Inputs.ToolResult_59.MatchingRate       :=  TO_UINT(_word);        // IW1232
            _word.%B0 := _data_in[3];
            _word.%B1 := _data_in[2];
            Inputs.ToolResult_59.MatchingRateMAX    :=  TO_UINT(_word);        // IW1234
            _word.%B0 := _data_in[5];
            _word.%B1 := _data_in[4];
            Inputs.ToolResult_59.MatchingRateMIN    :=  TO_UINT(_word);        // IW1236
            _word.%B0 := _data_in[7];
            _word.%B1 := _data_in[6];
            Inputs.ToolResult_59.LowerThreshold     :=  TO_UINT(_word);        // IW1238
            _word.%B0 := _data_in[9];
            _word.%B1 := _data_in[8];
            Inputs.ToolResult_59.UpperThreshold     :=  TO_UINT(_word);        // IW1240
            _word.%B0 := _data_in[11];
            _word.%B1 := _data_in[10];
            Inputs.ToolResult_59.DecimalPointPosition:=  TO_UINT(_word);       // IW1242
            _word.%B0 := _data_in[13];
            _word.%B1 := _data_in[12];
            Inputs.ToolResult_59.Data_1             :=  TO_UINT(_word);        // IW1244
            _word.%B0 := _data_in[15];
            _word.%B1 := _data_in[14];
            Inputs.ToolResult_59.Data_2             :=  TO_UINT(_word);        // IW1246
            _word.%B0 := _data_in[17];
            _word.%B1 := _data_in[16];
            Inputs.ToolResult_59.Data_3             :=  TO_UINT(_word);        // IW1248
                                                                                    // IW1250
            //***************************************************************

            //*************************ToolResult_60*************************
            _retVal := Siemens.Simatic.DistributedIO.ReadData((Config.HWIDs.HwID_ToolResult_60) ,_data_in);
            IF _retVal > WORD#0 THEN
                Messenger.Activate(UINT#1665, eAxoMessageCategory#Error);
                Status.Error.Id := UINT#1665;
                RETURN;
            END_IF;

            _word.%B0 := _data_in[1];
            _word.%B1 := _data_in[0];
            Inputs.ToolResult_60.MatchingRate       :=  TO_UINT(_word);        // IW1252
            _word.%B0 := _data_in[3];
            _word.%B1 := _data_in[2];
            Inputs.ToolResult_60.MatchingRateMAX    :=  TO_UINT(_word);        // IW1254
            _word.%B0 := _data_in[5];
            _word.%B1 := _data_in[4];
            Inputs.ToolResult_60.MatchingRateMIN    :=  TO_UINT(_word);        // IW1256
            _word.%B0 := _data_in[7];
            _word.%B1 := _data_in[6];
            Inputs.ToolResult_60.LowerThreshold     :=  TO_UINT(_word);        // IW1258
            _word.%B0 := _data_in[9];
            _word.%B1 := _data_in[8];
            Inputs.ToolResult_60.UpperThreshold     :=  TO_UINT(_word);        // IW1260
            _word.%B0 := _data_in[11];
            _word.%B1 := _data_in[10];
            Inputs.ToolResult_60.DecimalPointPosition:=  TO_UINT(_word);       // IW1262
            _word.%B0 := _data_in[13];
            _word.%B1 := _data_in[12];
            Inputs.ToolResult_60.Data_1             :=  TO_UINT(_word);        // IW1264
            _word.%B0 := _data_in[15];
            _word.%B1 := _data_in[14];
            Inputs.ToolResult_60.Data_2             :=  TO_UINT(_word);        // IW1266
            _word.%B0 := _data_in[17];
            _word.%B1 := _data_in[16];
            Inputs.ToolResult_60.Data_3             :=  TO_UINT(_word);        // IW1268
                                                                                    // IW1270
            //***************************************************************

            //*************************ToolResult_61*************************
            _retVal := Siemens.Simatic.DistributedIO.ReadData((Config.HWIDs.HwID_ToolResult_61) ,_data_in);
            IF _retVal > WORD#0 THEN
                Messenger.Activate(UINT#1666, eAxoMessageCategory#Error);
                Status.Error.Id := UINT#1666;
                RETURN;
            END_IF;

            _word.%B0 := _data_in[1];
            _word.%B1 := _data_in[0];
            Inputs.ToolResult_61.MatchingRate       :=  TO_UINT(_word);        // IW1272
            _word.%B0 := _data_in[3];
            _word.%B1 := _data_in[2];
            Inputs.ToolResult_61.MatchingRateMAX    :=  TO_UINT(_word);        // IW1274
            _word.%B0 := _data_in[5];
            _word.%B1 := _data_in[4];
            Inputs.ToolResult_61.MatchingRateMIN    :=  TO_UINT(_word);        // IW1276
            _word.%B0 := _data_in[7];
            _word.%B1 := _data_in[6];
            Inputs.ToolResult_61.LowerThreshold     :=  TO_UINT(_word);        // IW1278
            _word.%B0 := _data_in[9];
            _word.%B1 := _data_in[8];
            Inputs.ToolResult_61.UpperThreshold     :=  TO_UINT(_word);        // IW1280
            _word.%B0 := _data_in[11];
            _word.%B1 := _data_in[10];
            Inputs.ToolResult_61.DecimalPointPosition:=  TO_UINT(_word);       // IW1282
            _word.%B0 := _data_in[13];
            _word.%B1 := _data_in[12];
            Inputs.ToolResult_61.Data_1             :=  TO_UINT(_word);        // IW1284
            _word.%B0 := _data_in[15];
            _word.%B1 := _data_in[14];
            Inputs.ToolResult_61.Data_2             :=  TO_UINT(_word);        // IW1286
            _word.%B0 := _data_in[17];
            _word.%B1 := _data_in[16];
            Inputs.ToolResult_61.Data_3             :=  TO_UINT(_word);        // IW1288
                                                                                    // IW1290
            //***************************************************************

            //*************************ToolResult_62*************************
            _retVal := Siemens.Simatic.DistributedIO.ReadData((Config.HWIDs.HwID_ToolResult_62) ,_data_in);
            IF _retVal > WORD#0 THEN
                Messenger.Activate(UINT#1667, eAxoMessageCategory#Error);
                Status.Error.Id := UINT#1667;
                RETURN;
            END_IF;

            _word.%B0 := _data_in[1];
            _word.%B1 := _data_in[0];
            Inputs.ToolResult_62.MatchingRate       :=  TO_UINT(_word);        // IW1292
            _word.%B0 := _data_in[3];
            _word.%B1 := _data_in[2];
            Inputs.ToolResult_62.MatchingRateMAX    :=  TO_UINT(_word);        // IW1294
            _word.%B0 := _data_in[5];
            _word.%B1 := _data_in[4];
            Inputs.ToolResult_62.MatchingRateMIN    :=  TO_UINT(_word);        // IW1296
            _word.%B0 := _data_in[7];
            _word.%B1 := _data_in[6];
            Inputs.ToolResult_62.LowerThreshold     :=  TO_UINT(_word);        // IW1298
            _word.%B0 := _data_in[9];
            _word.%B1 := _data_in[8];
            Inputs.ToolResult_62.UpperThreshold     :=  TO_UINT(_word);        // IW1300
            _word.%B0 := _data_in[11];
            _word.%B1 := _data_in[10];
            Inputs.ToolResult_62.DecimalPointPosition:=  TO_UINT(_word);       // IW1302
            _word.%B0 := _data_in[13];
            _word.%B1 := _data_in[12];
            Inputs.ToolResult_62.Data_1             :=  TO_UINT(_word);        // IW1304
            _word.%B0 := _data_in[15];
            _word.%B1 := _data_in[14];
            Inputs.ToolResult_62.Data_2             :=  TO_UINT(_word);        // IW1306
            _word.%B0 := _data_in[17];
            _word.%B1 := _data_in[16];
            Inputs.ToolResult_62.Data_3             :=  TO_UINT(_word);        // IW1308
                                                                                    // IW1310
            //***************************************************************

            //*************************ToolResult_63*************************
            _retVal := Siemens.Simatic.DistributedIO.ReadData((Config.HWIDs.HwID_ToolResult_63) ,_data_in);
            IF _retVal > WORD#0 THEN
                Messenger.Activate(UINT#1668, eAxoMessageCategory#Error);
                Status.Error.Id := UINT#1668;
                RETURN;
            END_IF;

            _word.%B0 := _data_in[1];
            _word.%B1 := _data_in[0];
            Inputs.ToolResult_63.MatchingRate       :=  TO_UINT(_word);        // IW1312
            _word.%B0 := _data_in[3];
            _word.%B1 := _data_in[2];
            Inputs.ToolResult_63.MatchingRateMAX    :=  TO_UINT(_word);        // IW1314
            _word.%B0 := _data_in[5];
            _word.%B1 := _data_in[4];
            Inputs.ToolResult_63.MatchingRateMIN    :=  TO_UINT(_word);        // IW1316
            _word.%B0 := _data_in[7];
            _word.%B1 := _data_in[6];
            Inputs.ToolResult_63.LowerThreshold     :=  TO_UINT(_word);        // IW1318
            _word.%B0 := _data_in[9];
            _word.%B1 := _data_in[8];
            Inputs.ToolResult_63.UpperThreshold     :=  TO_UINT(_word);        // IW1320
            _word.%B0 := _data_in[11];
            _word.%B1 := _data_in[10];
            Inputs.ToolResult_63.DecimalPointPosition:=  TO_UINT(_word);       // IW1322
            _word.%B0 := _data_in[13];
            _word.%B1 := _data_in[12];
            Inputs.ToolResult_63.Data_1             :=  TO_UINT(_word);        // IW1324
            _word.%B0 := _data_in[15];
            _word.%B1 := _data_in[14];
            Inputs.ToolResult_63.Data_2             :=  TO_UINT(_word);        // IW1326
            _word.%B0 := _data_in[17];
            _word.%B1 := _data_in[16];
            Inputs.ToolResult_63.Data_3             :=  TO_UINT(_word);        // IW1328
                                                                                    // IW1330
            //***************************************************************

            //*************************ToolResult_64*************************
            _retVal := Siemens.Simatic.DistributedIO.ReadData((Config.HWIDs.HwID_ToolResult_64) ,_data_in);
            IF _retVal > WORD#0 THEN
                Messenger.Activate(UINT#1669, eAxoMessageCategory#Error);
                Status.Error.Id := UINT#1669;
                RETURN;
            END_IF;

            _word.%B0 := _data_in[1];
            _word.%B1 := _data_in[0];
            Inputs.ToolResult_64.MatchingRate       :=  TO_UINT(_word);        // IW1332
            _word.%B0 := _data_in[3];
            _word.%B1 := _data_in[2];
            Inputs.ToolResult_64.MatchingRateMAX    :=  TO_UINT(_word);        // IW1334
            _word.%B0 := _data_in[5];
            _word.%B1 := _data_in[4];
            Inputs.ToolResult_64.MatchingRateMIN    :=  TO_UINT(_word);        // IW1336
            _word.%B0 := _data_in[7];
            _word.%B1 := _data_in[6];
            Inputs.ToolResult_64.LowerThreshold     :=  TO_UINT(_word);        // IW1338
            _word.%B0 := _data_in[9];
            _word.%B1 := _data_in[8];
            Inputs.ToolResult_64.UpperThreshold     :=  TO_UINT(_word);        // IW1340
            _word.%B0 := _data_in[11];
            _word.%B1 := _data_in[10];
            Inputs.ToolResult_64.DecimalPointPosition:=  TO_UINT(_word);       // IW1342
            _word.%B0 := _data_in[13];
            _word.%B1 := _data_in[12];
            Inputs.ToolResult_64.Data_1             :=  TO_UINT(_word);        // IW1344
            _word.%B0 := _data_in[15];
            _word.%B1 := _data_in[14];
            Inputs.ToolResult_64.Data_2             :=  TO_UINT(_word);        // IW1346
            _word.%B0 := _data_in[17];
            _word.%B1 := _data_in[16];
            Inputs.ToolResult_64.Data_3             :=  TO_UINT(_word);        // IW1348
                                                                                    // IW1350
            //***************************************************************

            //*************************DeviceResultBits_2********************
            _retVal := Siemens.Simatic.DistributedIO.ReadData((Config.HWIDs.HwID_DeviceResultBits_2) ,_data_in);
            IF _retVal > WORD#0 THEN
                Messenger.Activate(UINT#1670, eAxoMessageCategory#Error);
                Status.Error.Id := UINT#1670;
                RETURN;
            END_IF;

            _word.%B0 := _data_in[1];
            _word.%B1 := _data_in[0];
            Inputs.DeviceResultBits_2.MasterNumber                  :=  TO_UINT(_word);        // IW1352

            Inputs.DeviceResultBits_2.Tool_17                       :=   _data_in[2].%X0;       // IB1354.0
            Inputs.DeviceResultBits_2.Tool_18                       :=   _data_in[2].%X1;       // IB1354.1
            Inputs.DeviceResultBits_2.Tool_19                       :=   _data_in[2].%X2;       // IB1354.2
            Inputs.DeviceResultBits_2.Tool_20                       :=   _data_in[2].%X3;       // IB1354.3
            Inputs.DeviceResultBits_2.Tool_21                       :=   _data_in[2].%X4;       // IB1354.4
            Inputs.DeviceResultBits_2.Tool_22                       :=   _data_in[2].%X5;       // IB1354.5
            Inputs.DeviceResultBits_2.Tool_23                       :=   _data_in[2].%X6;       // IB1354.6
            Inputs.DeviceResultBits_2.Tool_24                       :=   _data_in[2].%X7;       // IB1354.7
            Inputs.DeviceResultBits_2.Tool_25                       :=   _data_in[3].%X0;       // IB1355.0
            Inputs.DeviceResultBits_2.Tool_26                       :=   _data_in[3].%X1;       // IB1355.1
            Inputs.DeviceResultBits_2.Tool_27                       :=   _data_in[3].%X2;       // IB1355.2
            Inputs.DeviceResultBits_2.Tool_28                       :=   _data_in[3].%X3;       // IB1355.3
            Inputs.DeviceResultBits_2.Tool_29                       :=   _data_in[3].%X4;       // IB1355.4
            Inputs.DeviceResultBits_2.Tool_30                       :=   _data_in[3].%X5;       // IB1355.5
            Inputs.DeviceResultBits_2.Tool_31                       :=   _data_in[3].%X6;       // IB1355.6
            Inputs.DeviceResultBits_2.Tool_32                       :=   _data_in[3].%X7;       // IB1355.7
            Inputs.DeviceResultBits_2.Tool_33                       :=   _data_in[4].%X0;       // IB1356.0
            Inputs.DeviceResultBits_2.Tool_34                       :=   _data_in[4].%X1;       // IB1356.1
            Inputs.DeviceResultBits_2.Tool_35                       :=   _data_in[4].%X2;       // IB1356.2
            Inputs.DeviceResultBits_2.Tool_36                       :=   _data_in[4].%X3;       // IB1356.3
            Inputs.DeviceResultBits_2.Tool_37                       :=   _data_in[4].%X4;       // IB1356.4
            Inputs.DeviceResultBits_2.Tool_38                       :=   _data_in[4].%X5;       // IB1356.5
            Inputs.DeviceResultBits_2.Tool_39                       :=   _data_in[4].%X6;       // IB1356.6
            Inputs.DeviceResultBits_2.Tool_40                       :=   _data_in[4].%X7;       // IB1356.7
            Inputs.DeviceResultBits_2.Tool_41                       :=   _data_in[5].%X0;       // IB1357.0
            Inputs.DeviceResultBits_2.Tool_42                       :=   _data_in[5].%X1;       // IB1357.1
            Inputs.DeviceResultBits_2.Tool_43                       :=   _data_in[5].%X2;       // IB1357.2
            Inputs.DeviceResultBits_2.Tool_44                       :=   _data_in[5].%X3;       // IB1357.3
            Inputs.DeviceResultBits_2.Tool_45                       :=   _data_in[5].%X4;       // IB1357.4
            Inputs.DeviceResultBits_2.Tool_46                       :=   _data_in[5].%X5;       // IB1357.5
            Inputs.DeviceResultBits_2.Tool_47                       :=   _data_in[5].%X6;       // IB1357.6
            Inputs.DeviceResultBits_2.Tool_48                       :=   _data_in[5].%X7;       // IB1357.7
            Inputs.DeviceResultBits_2.Tool_49                       :=   _data_in[6].%X0;       // IB1358.0
            Inputs.DeviceResultBits_2.Tool_50                       :=   _data_in[6].%X1;       // IB1358.1
            Inputs.DeviceResultBits_2.Tool_51                       :=   _data_in[6].%X2;       // IB1358.2
            Inputs.DeviceResultBits_2.Tool_52                       :=   _data_in[6].%X3;       // IB1358.3
            Inputs.DeviceResultBits_2.Tool_53                       :=   _data_in[6].%X4;       // IB1358.4
            Inputs.DeviceResultBits_2.Tool_54                       :=   _data_in[6].%X5;       // IB1358.5
            Inputs.DeviceResultBits_2.Tool_55                       :=   _data_in[6].%X6;       // IB1358.6
            Inputs.DeviceResultBits_2.Tool_56                       :=   _data_in[6].%X7;       // IB1358.7
            Inputs.DeviceResultBits_2.Tool_57                       :=   _data_in[7].%X0;       // IB1359.0
            Inputs.DeviceResultBits_2.Tool_58                       :=   _data_in[7].%X1;       // IB1359.1
            Inputs.DeviceResultBits_2.Tool_59                       :=   _data_in[7].%X2;       // IB1359.2
            Inputs.DeviceResultBits_2.Tool_60                       :=   _data_in[7].%X3;       // IB1359.3
            Inputs.DeviceResultBits_2.Tool_61                       :=   _data_in[7].%X4;       // IB1359.4
            Inputs.DeviceResultBits_2.Tool_62                       :=   _data_in[7].%X5;       // IB1359.5
            Inputs.DeviceResultBits_2.Tool_63                       :=   _data_in[7].%X6;       // IB1359.6
            Inputs.DeviceResultBits_2.Tool_64                       :=   _data_in[7].%X7;       // IB1359.7

            //***************************************************************

            //*************INITIALIZATION*************
            RestoreTask.Run(THIS);
            TriggerTask.Run(THIS);
            ChangeProgramTask.Run(THIS);

            //****************************************

            //********************Diagnostics*********
            HardwareDiagnosticsTask.Run(THIS,Config.HWIDs.HW_Device);
            IF Inputs.CommandStatusBits.Error THEN
                Messenger.Activate(UINT#1800 + Inputs.DeviceStatusWords.ErrorNo, eAxoMessageCategory#Error);
                Status.Error.Id := UINT#1800 + Inputs.DeviceStatusWords.ErrorNo;
            ELSIF Inputs.CommandStatusBits.Warning THEN
                Messenger.Activate(UINT#400 + Inputs.DeviceStatusWords.WarningNo, eAxoMessageCategory#Warning);
                Status.Error.Id := UINT#400 + Inputs.DeviceStatusWords.WarningNo;
            END_IF;
            //****************************************

            //*************RESTORE********************
            RestoreTask.IsDisabled := FALSE;
            IF RestoreTask.Execute(THIS) THEN
                THIS.Restore();
            END_IF;
            //****************************************

            //*************TriggerTask**************
            TriggerTask.SetIsDisabled(FALSE);
            IF TriggerTask.StartTriggered() THEN
                Status.Action.Id :=  UINT#100;
            END_IF;
            Messenger.ActivateOnCondition(ULINT#100,TriggerTask.IsBusy(), eAxoMessageCategory#Info);
            Messenger.ActivateOnCondition(ULINT#101,TriggerTask.IsDone(), eAxoMessageCategory#Info);
            IF TriggerTask.Execute(THIS) THEN
                IF _progress = 0 THEN
                    _resultUpdateComplete := Inputs.CommandStatusBits.ResultUpdateComplete;
                    _resultNo := Inputs.DeviceStatusWords.ResultNo;
                    Outputs.CommandControl.TriggerRequest                               := FALSE;
                    Outputs.CommandControl.MasterRegistrationRequest                    := FALSE;
                    Outputs.CommandControl.ProgramSwitchingRequest                      := FALSE;
                    Outputs.CommandControl.WarningClearRequest                          := FALSE;
                    Outputs.CommandControl.StatisticsResetRequest                       := FALSE;
                    Outputs.CommandControl.BufferClearRequest                           := FALSE;
                    Outputs.CommandControl.SdCardSavingStopRequest                      := FALSE;
                    Outputs.CommandControl.SettingValueChangeRequest                    := FALSE;
                    Outputs.CommandControl.ResultAcquisitionCompleteNotification        := FALSE;
                    Status.Error.Id := UINT#0;
                    TaskMessenger.Restore();
                    THIS.CallTimers(FALSE);
                    _progress := 300;
                END_IF;
                // TriggerTask running: waiting for the raising of the 'TriggerReady' signal.
                IF _progress = 300 THEN
                    IF _infoTimer.output THEN
                        TaskMessenger.Activate( UINT#500, eAxoMessageCategory#Potential);
                        Status.Error.Id :=      UINT#500;
                    END_IF;

                    IF Inputs.CommandStatusBits.TriggerReady THEN
                        THIS.CallTimers(FALSE);
                        _progress := 301;
                    END_IF;
                END_IF;
                // TriggerTask running: waiting for the raising of the 'TriggerResponse' signal.
                IF _progress = 301 THEN
                    IF _infoTimer.output THEN
                        TaskMessenger.Activate( UINT#501, eAxoMessageCategory#Potential);
                        Status.Error.Id :=      UINT#501;
                    END_IF;

                    Outputs.CommandControl.TriggerRequest := TRUE;

                    IF Inputs.CommandStatusBits.TriggerResponse THEN
                        THIS.CallTimers(FALSE);
                        _progress := 302;
                    END_IF;
                END_IF;
                // TriggerTask running: waiting for the raising of the 'BUSY' signal.
                IF _progress = 302 THEN
                    IF _infoTimer.output THEN
                        TaskMessenger.Activate( UINT#502, eAxoMessageCategory#Potential);
                        Status.Error.Id :=      UINT#502;
                    END_IF;

                    IF Inputs.CommandStatusBits.BUSY THEN
                        THIS.CallTimers(FALSE);
                        _progress := 303;
                    END_IF;
                END_IF;
                // TriggerTask running: waiting for the raising of the 'ImagingStatus' signal.
                IF _progress = 303 THEN
                    IF _infoTimer.output THEN
                        TaskMessenger.Activate( UINT#503, eAxoMessageCategory#Potential);
                        Status.Error.Id :=      UINT#503;
                    END_IF;

                    IF TRUE OR Inputs.CommandStatusBits.ImagingStatus THEN
                        THIS.CallTimers(FALSE);
                        _progress := 304;
                    END_IF;
                END_IF;
                // TriggerTask running: waiting for the falling of the 'BUSY' signal.
                IF _progress = 304 THEN
                    IF _infoTimer.output THEN
                        TaskMessenger.Activate( UINT#504, eAxoMessageCategory#Potential);
                        Status.Error.Id :=      UINT#504;
                    END_IF;

                    Outputs.CommandControl.TriggerRequest := FALSE;

                    IF NOT Inputs.CommandStatusBits.BUSY THEN
                        THIS.CallTimers(FALSE);
                        _progress := 305;
                    END_IF;
                END_IF;
                // TriggerTask running: waiting for the change of the 'ResultUpdateComplete' signal.
                IF _progress = 305 THEN
                    IF _infoTimer.output THEN
                        TaskMessenger.Activate( UINT#505, eAxoMessageCategory#Potential);
                        Status.Error.Id :=      UINT#505;
                    END_IF;

                    IF Inputs.CommandStatusBits.ResultUpdateComplete <> _resultUpdateComplete THEN
                        THIS.CallTimers(FALSE);
                        _progress := 306;
                    END_IF;
                END_IF;
                // TriggerTask running: waiting for the raising of the 'ResultAvailable' signal.
                IF _progress = 306 THEN
                    IF _infoTimer.output THEN
                        TaskMessenger.Activate( UINT#506, eAxoMessageCategory#Potential);
                        Status.Error.Id :=      UINT#506;
                    END_IF;

                    IF Inputs.CommandStatusBits.ResultAvailable THEN
                        THIS.CallTimers(FALSE);
                        _progress := 307;
                    END_IF;
                END_IF;
                // TriggerTask running: waiting for the incrementation of the 'ResultNo' signal.
                IF _progress = 307 THEN
                    IF _infoTimer.output THEN
                        TaskMessenger.Activate( UINT#507, eAxoMessageCategory#Potential);
                        Status.Error.Id :=      UINT#507;
                    END_IF;

                    IF Inputs.DeviceStatusWords.ResultNo > _resultNo THEN
                        THIS.CallTimers(FALSE);
                        _progress := 308;
                    END_IF;
                END_IF;
                // TriggerTask finished.
                IF _progress = 308 THEN
                    TriggerTask.DoneWhen(TRUE);
                    _progress := 0;
                END_IF;

                THIS.CallTimers(TRUE);

                TriggerTask.ThrowWhen(_errorTimer.output);
                Status.Action.Id := TO_UINT(_progress);
                TriggerTask.ThrowWhen(TriggerTask.Duration >= Config.TaskTimeout AND Config.TaskTimeout > T#0s ,'<#TriggerTask timeout.#>');
            END_IF;
            IF TriggerTask.DoneReached() THEN
                Status.Action.Id :=  UINT#101;
                Status.Error.Id :=  UINT#0;
            ELSIF TriggerTask.ErrorOccured() THEN
                Status.Action.Id :=  UINT#10000;
                Status.Error.Id  :=  UINT#10000;
            ELSIF TriggerTask.AbortTriggered()THEN
                Status.Action.Id :=  UINT#10001;
                Status.Error.Id  :=  UINT#10001;
            END_IF;
            Messenger.ActivateOnCondition(ULINT#10000,TriggerTask.HasError(), eAxoMessageCategory#Error);
            Messenger.ActivateOnCondition(ULINT#10001,TriggerTask.IsAborted(), eAxoMessageCategory#Info);
            Messenger.ActivateOnCondition(ULINT#102,TriggerTask.RestoreTriggered() , eAxoMessageCategory#Info);
            IF TriggerTask.RestoreTriggered() AND _progress >= 300 AND _progress <= 309  THEN
                Status.Action.Id :=  UINT#102;
                _progress := 0;
            END_IF;
            //**************************************************

            //*************ChangeProgramTask***************
            ChangeProgramTask.SetIsDisabled(FALSE);
            IF ChangeProgramTask.StartTriggered() THEN
                Status.Action.Id :=  UINT#110;
            END_IF;
            Messenger.ActivateOnCondition(ULINT#110,ChangeProgramTask.IsBusy(), eAxoMessageCategory#Info);
            Messenger.ActivateOnCondition(ULINT#111,ChangeProgramTask.IsDone(), eAxoMessageCategory#Info);
            IF ChangeProgramTask.Execute(THIS) THEN
                IF _progress = 0 THEN
                    THIS.ClearProgressRoot();
                    THIS.AddProgressToRoot(0);

                    Outputs.CommandControl.TriggerRequest                               := FALSE;
                    Outputs.CommandControl.MasterRegistrationRequest                    := FALSE;
                    Outputs.CommandControl.ProgramSwitchingRequest                      := FALSE;
                    Outputs.CommandControl.WarningClearRequest                          := FALSE;
                    Outputs.CommandControl.StatisticsResetRequest                       := FALSE;
                    Outputs.CommandControl.BufferClearRequest                           := FALSE;
                    Outputs.CommandControl.SdCardSavingStopRequest                      := FALSE;
                    Outputs.CommandControl.SettingValueChangeRequest                    := FALSE;
                    Outputs.CommandControl.ResultAcquisitionCompleteNotification        := FALSE;
                    Status.Error.Id := UINT#0;
                    TaskMessenger.Restore();
                    THIS.CallTimers(FALSE);

                    _ProgChangeInterrupted := FALSE;
                    _progress := 310;
                END_IF;
                // ChangeProgramTask running: checking the program number.
                IF _progress = 310 THEN
                    THIS.AddProgressToRoot(310);

                    IF _programNumber <= Config.MaxProgramNumber THEN
                        THIS.CallTimers(FALSE);
                        _progress := 311;
                    ELSE
                        TaskMessenger.Activate( UINT#510, eAxoMessageCategory#Potential);
                        Status.Error.Id :=      UINT#510;
                    END_IF;
                END_IF;

                 // ChangeProgramTask running: if 'ProgramSwitchingResponse' signal is true, finish previous change.
                IF _progress = 311 THEN
                    THIS.AddProgressToRoot(311);

                    IF _infoTimer.output THEN
                        TaskMessenger.Activate( UINT#511, eAxoMessageCategory#Potential);
                        Status.Error.Id :=      UINT#511;
                    END_IF;

                    // Do not cancel (1 → 0) [Program switching request] before [Program switching response] changes from
                    // 0 to 1. The program may not be able to switch correctly.
                    // When [Program switching request] was canceled (1 → 0) before [Program switching response] changes
                    // from 0 to 1, execute (0 → 1) [Program switching request] and cancel (1 → 0) it again.

                    IF Inputs.CommandStatusBits.ProgramSwitchingResponse THEN
                        THIS.CallTimers(FALSE);
                        _ProgChangeInterrupted := TRUE;
                        _progress := 312; // ACK PREVIOUS CHANGE
                    ELSE
                        THIS.CallTimers(FALSE);
                        _progress := 314; // Continue to change program
                    END_IF;
                END_IF;

                 // evaluated before 312 => +1 plc cycle
                 // ChangeProgramTask running: check if is not Busy, due to interrupted by previous program switching
                IF _progress = 313 THEN
                    THIS.AddProgressToRoot(313);
                    IF _infoTimer.output THEN
                        TaskMessenger.Activate( UINT#513, eAxoMessageCategory#Potential);
                        Status.Error.Id :=      UINT#513;
                    END_IF;

                    Outputs.CommandControl.ProgramSwitchingRequest     := FALSE;
                    IF NOT Inputs.CommandStatusBits.BUSY  THEN
                        THIS.CallTimers(FALSE);
                        _progress := 311; // +1 plc cycle to check ProgramSwitchingResponse
                    END_IF;
                END_IF;

                // ChangeProgramTask running: set [program switching request] to 1 due to interupted by previous program switching
                IF _progress = 312 THEN
                        THIS.AddProgressToRoot(312);
                    IF _infoTimer.output THEN
                        TaskMessenger.Activate( UINT#513, eAxoMessageCategory#Potential);
                        Status.Error.Id :=      UINT#513;
                    END_IF;

                    Outputs.CommandControl.ProgramSwitchingRequest     := TRUE;
                    Outputs.CommandControl.ProgramNo                   := UINT#0; // Reset program number
                    IF TRUE THEN
                        THIS.CallTimers(FALSE);
                        _progress := 313; //+1 plc cycle to wait for falling edge
                    END_IF;
                END_IF;

                // ChangeProgramTask running: check if is needed to change program, if current program number is not equal to target program number, continue to change, otherwise skip to the end.
                IF _progress = 314 THEN
                        THIS.AddProgressToRoot(314);
                    IF _infoTimer.output THEN
                        TaskMessenger.Activate( UINT#511, eAxoMessageCategory#Potential);
                        Status.Error.Id :=      UINT#511;
                    END_IF;

                    // IF _programNumber = Inputs.DeviceStatusWords.CurrentProgramNo THEN // is is equel, skipt to the end, otherwise wait for the change
                    //     THIS.CallTimers(FALSE);
                    //     _progress := 317;
                    // ELSE
                        THIS.CallTimers(FALSE);
                        _progress := 315;
                    // END_IF;
                END_IF;

                // ChangeProgramTask running: set 'ProgramSwitchingRequest' and wait for 'ProgramSwitchingResponse' signal.
                IF _progress = 315 THEN
                    THIS.AddProgressToRoot(315);
                    IF _infoTimer.output THEN
                        TaskMessenger.Activate( UINT#512, eAxoMessageCategory#Potential);
                        Status.Error.Id :=      UINT#512;
                    END_IF;

                    Outputs.CommandControl.ProgramNo                := _programNumber;
                    Outputs.CommandControl.ProgramSwitchingRequest  := TRUE;

                    IF Inputs.CommandStatusBits.ProgramSwitchingResponse THEN
                        THIS.CallTimers(FALSE);
                        _progress := 316;
                    END_IF;
                END_IF;

                // ChangeProgramTask running: waiting for the falling of the 'ProgramSwitchingResponse' signal, when 'ProgramSwitchingRequest' is reset.
                IF _progress = 316 THEN
                    THIS.AddProgressToRoot(316);
                    IF _infoTimer.output THEN
                        TaskMessenger.Activate( UINT#513, eAxoMessageCategory#Potential);
                        Status.Error.Id :=      UINT#513;
                    END_IF;

                    Outputs.CommandControl.ProgramSwitchingRequest  := FALSE;
                    Outputs.CommandControl.ProgramNo := UINT#0; // Reset program number , accoding documentation

                    IF NOT Inputs.CommandStatusBits.ProgramSwitchingResponse THEN
                        THIS.CallTimers(FALSE);
                        _progress := 317;
                    END_IF;
                END_IF;

                // ChangeProgramTask running: validate that program is selected successfully and other control signals are right,
                IF _progress = 318 THEN
                    THIS.AddProgressToRoot(318);
                    IF _infoTimer.output THEN
                        TaskMessenger.Activate( UINT#513, eAxoMessageCategory#Potential);
                        Status.Error.Id :=      UINT#513;
                    END_IF;

                    IF  NOT Inputs.CommandStatusBits.ProgramSwitchingResponse
                        AND  NOT Inputs.CommandStatusBits.BUSY
                        AND ( Inputs.DeviceStatusWords.CurrentProgramNo = _programNumber)
                    THEN
                        THIS.CallTimers(FALSE);
                        _progress := 319;
                    END_IF;
                END_IF;

                // ChangeProgramTask running: validate that program is selected successfully,
                IF _progress = 317 THEN
                    THIS.AddProgressToRoot(317);
                    IF _infoTimer.output THEN
                        TaskMessenger.Activate( UINT#513, eAxoMessageCategory#Potential);
                        Status.Error.Id :=      UINT#513;
                    END_IF;

                    IF (_programNumber = Inputs.DeviceStatusWords.CurrentProgramNo) THEN
                        THIS.CallTimers(FALSE);
                        _progress := 318; //+1 plc cycle to check the status after program change
                    END_IF;
                END_IF;

                // ChangeProgramTask finished.
                IF _progress = 319 THEN
                        THIS.AddProgressToRoot(319);
                    ChangeProgramTask.DoneWhen(TRUE);
                    _progress := 0;
                END_IF;

                THIS.CallTimers(TRUE);

                ChangeProgramTask.ThrowWhen(Inputs.CommandStatusBits.ProgramSwitchingFailed,'<#Attempt to change the program failed.#>');
                ChangeProgramTask.ThrowWhen(_errorTimer.output);
                Status.Action.Id := TO_UINT(_progress);
                ChangeProgramTask.ThrowWhen(ChangeProgramTask.Duration >= Config.TaskTimeout AND Config.TaskTimeout > T#0s ,'<#ChangeProgramTask timeout.#>');
            END_IF;
            IF ChangeProgramTask.DoneReached() THEN
                Status.Action.Id :=  UINT#111;
                Status.Error.Id :=  UINT#0;
            ELSIF ChangeProgramTask.ErrorOccured() THEN
                Status.Action.Id :=  UINT#10010;
                Status.Error.Id  :=  UINT#10010;
            ELSIF ChangeProgramTask.AbortTriggered()THEN
                Status.Action.Id :=  UINT#10011;
                Status.Error.Id  :=  UINT#10011;
            END_IF;
            Messenger.ActivateOnCondition(ULINT#10010,ChangeProgramTask.HasError(), eAxoMessageCategory#Error);
            Messenger.ActivateOnCondition(ULINT#10011,ChangeProgramTask.IsAborted(), eAxoMessageCategory#Info);
            Messenger.ActivateOnCondition(ULINT#112,ChangeProgramTask.RestoreTriggered() , eAxoMessageCategory#Info);
            IF ChangeProgramTask.RestoreTriggered() AND _progress >= 310 AND _progress <= 329  THEN
                Status.Action.Id :=  UINT#112;
                _progress := 0;
            END_IF;
            //**************************************************

            //***********Update outputs ****************
            _data_out_12[0].%X0                  :=      Outputs.CommandControl.TriggerRequest;                        //  QB0.0
            _data_out_12[0].%X1                  :=      Outputs.CommandControl.MasterRegistrationRequest;             //  QB0.1
            _data_out_12[0].%X2                  :=      Outputs.CommandControl.ProgramSwitchingRequest;               //  QB0.2
            _data_out_12[0].%X3                  :=      Outputs.CommandControl.WarningClearRequest;                   //  QB0.3
            _data_out_12[0].%X4                  :=      Outputs.CommandControl.StatisticsResetRequest;                //  QB0.4
            _data_out_12[0].%X5                  :=      Outputs.CommandControl.BufferClearRequest;                    //  QB0.5
            _data_out_12[0].%X6                  :=      Outputs.CommandControl.SdCardSavingStopRequest;               //  QB0.6
            _data_out_12[0].%X7                  :=      Outputs.CommandControl.SettingValueChangeRequest;             //  QB0.7
            _data_out_12[2].%X0                  :=      Outputs.CommandControl.ResultAcquisitionCompleteNotification; //  QB2.0

            _word                                :=      TO_WORD(Outputs.CommandControl.ProgramNo);                    //  QW4
            _data_out_12[4]                      :=      _word.%B1;                                             //  QW4
            _data_out_12[5]                      :=      _word.%B0;                                             //  QW4

            _data_out_12[6]                      :=      Outputs.CommandControl.Function_1.%B1;                         //  QW6
            _data_out_12[7]                      :=      Outputs.CommandControl.Function_1.%B0;                         //  QW6

            _data_out_12[8]                      :=      Outputs.CommandControl.Function_2.%B3;                         //  QD8
            _data_out_12[9]                      :=      Outputs.CommandControl.Function_2.%B2;                         //  QD8
            _data_out_12[10]                     :=      Outputs.CommandControl.Function_2.%B1;                         //  QD8
            _data_out_12[11]                     :=      Outputs.CommandControl.Function_2.%B0;                         //  QD8

            _retVal := Siemens.Simatic.DistributedIO.WriteData((Config.HWIDs.HwID_CommandControl),_data_out_12);
            IF _retVal > WORD#0 THEN
                Messenger.Activate(UINT#1701, eAxoMessageCategory#ProgrammingError);
                Status.Error.Id := UINT#1701;
                RETURN;
            END_IF;
            //******************************************

        END_METHOD

        METHOD PUBLIC Trigger : IAxoTaskState
            Trigger := TriggerTask.Invoke(THIS);
        END_METHOD

        METHOD PUBLIC ChangeProgram : IAxoTaskState
            VAR_INPUT
                inProgramNumber : UINT;
            END_VAR

            // different program loaded in HW - restore task to be able to run it again
            IF ( inProgramNumber <> Inputs.DeviceStatusWords.CurrentProgramNo ) && ChangeProgramTask.IsDone() THEN
                ChangeProgramTask.Restore();
            END_IF;
